FUNCTION Convert_WORD_TO_WORD : BOOL
VAR_INPUT
	in : WORD;
	out : REFERENCE TO WORD;
END_VAR

out := in;
Convert_WORD_TO_WORD := TRUE;

END_FUNCTION

(* stored: Version 1.1.0.1, ProductVersion 3.1.4024.12
   POU Convert_WORD_TO_WORD: Id {5ae92396-4a21-4c22-81b2-4bfa3004f351}, SpecialFunc None *)
